{attribute 'GeneratedUsingTerminal: AT2025-0250-0022'}
{attribute addProperty BoxType "AT2025-0250-0022"}
{attribute addProperty Id "A_0075_AT2000_5250_0019_AT2000_5250AT2000_33A3DF1B80"}
{attribute addProperty CRC "3901712034"}
{attribute addProperty Size "80"}
TYPE A_0063_AT2025_0250_0022_AT2025_0250_E88F66A2 EXTENDS AT2025_2EA6C9BF :
STRUCT
	{attribute addProperty Name "A_0075_AT2000_5250_0019_AT2000_5250"}
	A_0075_AT2000_5250_0019_AT2000_5250 : AT2000_33A3DF1B;
END_STRUCT
END_TYPE

(* stored: Version 1.2.0.0, ProductVersion 3.1.4024.9
   DUT A_0063_AT2025_0250_0022_AT2025_0250_E88F66A2: Id {a25779f1-3303-4277-b28d-903170dbea12} *)
